{attribute 'qualified_only'}
{attribute 'strict'}
{attribute 'to_string'}
TYPE E_StationResultStatus :
(
    NotTested := 0,
    Pass := 10,
    Fail := 20
);
END_TYPE

(* stored: Version 1.1.0.1, ProductVersion 3.1.4026.18
   DUT E_StationResultStatus: Id {42e92727-80eb-4f9a-8d59-5d437f39e057} *)
